// TIA Portal V20 export
TYPE "typeEm1Monitoring"
// stored: Access Published, Namespace Unit1
   STRUCT
      jobinterface { ExternalWritable := 'False'} : "Unit1.typeEm1MonitoringJobInterface";
      cmStatus { ExternalWritable := 'False'} : "Unit1.typeEm1MonitoringCmStatus";
      UserDefine { ExternalWritable := 'False'} : "Unit1.typeEm1MonitoringUserDefine";
   END_STRUCT;
END_TYPE
